PROGRAM MAIN
VAR
	work_number	: ULINT;
	act_dc_time : T_DCTIME64;
	dc_task_time : T_DCTIME64;
	dc_tick_time : T_DCTIME64;
	diff_time : T_DCTIME64;
	fbConvertDcTimeToPos : ConvertDcTimeToPos;
	position_at_task_start_point : LREAL;
	position_diff : LREAL;
	dc_time_array : ARRAY [0..1] OF T_DCTIME32;
	
	fb_timezone_info : FB_GetTimeZoneInformation := (bExecute := TRUE);
	event_messages : ARRAY [1..3] OF STRING;
	
	fbPower1:mc_power;
	fbPower2:mc_power;
	fbStop	: MC_Stop;
	fbGearOut : MC_GearOut;
	fbReset	: MC_Reset;
	
	stop_job : FB_Executor;
	basic_job : FB_Executor;
	demo_job : FB_Executor;
	gear_in_job : FB_Executor;
	gear_out_job : FB_Executor;
	init_pos_job : FB_Executor;
	jog_plus_job : FB_Executor;
	jog_minus_job : FB_Executor;
	fb_observer : FB_Observer;
	job_reset : BOOL;
	
	mc_power_future_creator: FutureMCPowerCreator;
	mc_reset_future_creator: FutureMCResetCreator;
	mc_set_position_future_creator: FutureMCSetPositionCreator;
	mc_inching_future_creator : FutureMCInchingCreator;
	mc_gear_in_future_creator : FutureMCGearInCreator;
	mc_gear_out_future_creator : FutureMCGearOutCreator;
	mc_move_rel_future_creator : FutureMCMoveRelativeCreator;
	mc_move_abs_future_creator : FutureMCMoveAbsoluteCreator;
	mc_move_velocity_future_creator: FutureMCMoveVelocityCreator;
	mc_stop_future_creator: FutureMCStopCreator;
	sleep_creator : FutureSleepCreator;

	
	iState:UINT;
	stopState : UINT;
	stAxis1:axis_ref;
	stAxis2:axis_ref;
	bStart: BOOL;
	bJogPlus: BOOL;
	bJogMinus: BOOL;
	bPower: BOOL;
	_bPower :BOOL;
	bPowerOn : BOOL;
	iPowerState : UINT;
	bReset:BOOL;
	bError:BOOL;
	bAllAxisPowerOn: BOOL;
	bInsync:BOOL;
	create_container: INT;
	boot_up : BOOL := TRUE;
	i: UINT;
	
	quit: INT;	
END_VAR

// Update state data for axis_ref.Status structure.
stAxis1.ReadStatus();
stAxis2.ReadStatus();

act_dc_time := F_GetActualDcTime64();
dc_task_time := F_GetCurDcTaskTime64();
dc_tick_time := F_GetCurDcTickTime64();

MEMCPY(ADR(dc_time_array), ADR(dc_task_time), SIZEOF(dc_task_time));

fbConvertDcTimeToPos(nAxisId := 1, nSubIdx := 16#10000, dcTime := dc_time_array[0] + 300000);
position_at_task_start_point := fbConvertDcTimeToPos.fPosition;
position_diff := stAxis1.NcToPlc.ActPos - fbConvertDcTimeToPos.fPosition;

diff_time := act_dc_time - dc_task_time;

IF boot_up THEN
	(*
	Initial setting at the time of starting PLC.
	*)
	
	// Creating basic running job container instance
	basic_job.create_container(ContainerType.PARALLEL_QUEUE, 'BASIC');
	// Enable continuous mode : Continue running job after all queued jobs are purged.
	basic_job.continuous_mode := TRUE;
	// Set top level job name
	basic_job.id := 'M1';
	// Set observer object: for event logging, IoT
	basic_job.job_event_reporter := fb_observer;
	// Create position initialization job.
	JobCreate_PosInit(init_pos_job);
	// Create gear-in job.
	JobCreate_GearIn(gear_in_job);
	// Create demo job.
	JobCreateDemo(demo_job);
	// Create inching job
	mc_inching_future_creator.set_parameters(stAxis2, TRUE,1 , 100);
	jog_plus_job.create_future(mc_inching_future_creator,'JOG_PLUS');
	
	mc_inching_future_creator.set_parameters(stAxis2, FALSE, 1, 100);		
	jog_minus_job.create_future(mc_inching_future_creator,'JOG_MINUS');

	boot_up := FALSE;
END_IF

// Power control
// Power off after gear decoupled and job unlinked.

IF NOT bPower THEN
	CASE stopState OF
		0: // Forced stop if any jobs are working.
			IF bPowerOn THEN
				IF stAxis1.Status.HasJob THEN
					fbStop(Axis := stAxis1, Execute := TRUE);
				ELSE
					fbStop(Axis := stAxis1, Execute := FALSE);
					IF NOT fbStop.Busy THEN
						stopState := 1;
					END_IF
				END_IF
			END_IF
		1: // make job state abort
			IF basic_job.abort() THEN
				stopState := 2;	
			END_IF
		2: // Decouple stAxis2 from stAxis1.
			IF stAxis2.Status.Coupled THEN
				fbGearOut(Slave := stAxis2,Execute := TRUE);
			ELSE
				fbGearOut(Slave := stAxis2,Execute := FALSE);
				stopState := 3;
			END_IF
		3: // Unlink machie jobs and reset state machine. 
			IF basic_job.reset(FALSE) THEN
				IF basic_job.init() THEN
					bPowerOn := FALSE;
					bStart := FALSE;
					stopState := 0;
					iState := 0;
				END_IF
			END_IF	
	END_CASE
END_IF

IF bPower AND NOT _bPower THEN
	bPowerOn := TRUE;
END_IF

_bPower := bPower;

fbPower1(Axis := stAxis1, Enable := bPowerOn, Enable_Positive := TRUE, Enable_Negative := TRUE, Override := 100.0);
fbPower2(Axis := stAxis2, Enable := bPowerOn, Enable_Positive := TRUE, Enable_Negative := TRUE, Override := 100.0);

CASE iState OF
	0: // Position reset after Power ON
		IF fbPower1.Status AND fbPower2.Status THEN
			init_pos_job.init();
			basic_job.children.append_job(init_pos_job);
			iState := 1;
		END_IF
	1: // Vacant
		IF init_pos_job.done THEN
			iState := 2;
		END_IF
	2: // Adjustment coupling position between each gear, and to be start.
		IF bJogPlus THEN
			IF jog_plus_job.init() THEN
				basic_job.children.append_job(jog_plus_job);
				bJogPlus := FALSE;				
			END_IF
		END_IF
		
		IF bJogMinus THEN
			IF jog_minus_job.init() THEN
				basic_job.children.append_job(jog_minus_job);
				bJogMinus := FALSE;				
			END_IF
		END_IF

		IF bStart THEN
				IF NOT stAxis2.Status.Coupled THEN
					IF gear_in_job.init() THEN
						basic_job.children.append_job(gear_in_job);
						iState := 3;
					END_IF
				ELSE
					iState := 3;
				END_IF
		END_IF
	3: // Setting working job ID into demo_job instance and append it as machine job.
		IF demo_job.init() THEN
			work_number := work_number + 1;
			demo_job.id := TO_STRING(work_number);
			basic_job.children.append_job(demo_job);
			iState := 4;
		END_IF
	4: // Decision to finish or to rerun demo_job by Start button.
		IF demo_job.done THEN
			IF bStart THEN
				iState := 3;
			ELSE
				iState := 1;
			END_IF
		END_IF
END_CASE

basic_job.execute();

bError := basic_job.nErrorID <> 0;

IF bReset THEN
	IF basic_job.error_reset() THEN
		IF basic_job.resume() THEN
			bReset := FALSE;
		END_IF
	END_IF 
END_IF

fbReset(Axis := stAxis1, Execute := bReset);
fbReset(Axis := stAxis2, Execute := bReset);


IF basic_job.ready THEN
	basic_job.start();
END_IF

// Event string

IF fb_observer.job_event_report.new_state = TO_STRING(E_FutureExecutionState.process) THEN
	event_messages[1] := SYSTEMTIME_TO_STRING(FILETIME64_TO_SYSTEMTIME(fb_observer.job_event_report.record_time));
	event_messages[2] := fb_observer.job_event_report.future_name;
	event_messages[3] := fb_observer.job_event_report.job_id;
END_IF

METHOD Execution : BOOL
VAR_INPUT
	main_job : REFERENCE TO FB_Executor;
	bStart : BOOL := TRUE;
END_VAR
Execution := main_job.execute();

IF main_job.ready THEN
	main_job.start();
END_IF

IF bStart THEN
	main_job.start();
END_IF
END_METHOD

METHOD JobCreate_GearIn : BOOL
VAR_INPUT
	job : REFERENCE TO FB_Executor;
END_VAR
// Gear In
mc_gear_in_future_creator.set_parameters(stAxis1, stAxis2);
job.create_future(mc_gear_in_future_creator,'Gear IN');
END_METHOD

METHOD JobCreate_GearOut : BOOL
VAR_INPUT
	job : REFERENCE TO FB_Executor;
END_VAR
// Gear In
mc_gear_out_future_creator.set_parameters(stAxis2);
job.create_future(mc_gear_out_future_creator,'Gear OUT');
END_METHOD

METHOD JobCreate_PosInit : BOOL
VAR_INPUT
	job : REFERENCE TO FB_Executor;
END_VAR
VAR
	_job_temp	: REFERENCE TO FB_Executor; // reference to job object for working.
END_VAR
job.create_container(ContainerType.PARALLEL, 'INIT_POS');
// position set to 0
mc_set_position_future_creator.set_parameters(stAxis1, 0);
_job_temp REF= job.children.create_job(mc_set_position_future_creator,'AXIS1_POS_INIT');

mc_set_position_future_creator.set_parameters(stAxis2, 0);
_job_temp REF= job.children.create_job(mc_set_position_future_creator,'AXIS2_POS_INIT');
END_METHOD

METHOD JobCreate_Power : BOOL
VAR_INPUT
	power_on_job : REFERENCE TO FB_Executor;
	power_off_job : REFERENCE TO FB_Executor;
END_VAR
VAR
	_job_temp	: REFERENCE TO FB_Executor; // reference to job object for working.
END_VAR
power_on_job.create_container(ContainerType.PARALLEL, 'POWER_ON');
power_off_job.create_container(ContainerType.PARALLEL, 'POWER_OFF');
// position set to 0
mc_power_future_creator.set_parameters(stAxis1, TRUE);
power_on_job.children.create_job(mc_power_future_creator,'AXIS1_POWER_ON');
mc_power_future_creator.set_parameters(stAxis2, TRUE);
power_on_job.children.create_job(mc_power_future_creator,'AXIS2_POWER_ON');

mc_power_future_creator.set_parameters(stAxis1, FALSE);
power_off_job.children.create_job(mc_power_future_creator,'AXIS1_POWER_OFF');
mc_power_future_creator.set_parameters(stAxis2, FALSE);
power_off_job.children.create_job(mc_power_future_creator,'AXIS2_POWER_OFF');
END_METHOD

METHOD JobCreate_Stop : BOOL
VAR_INPUT
	job : REFERENCE TO FB_Executor;
END_VAR
mc_stop_future_creator.set_parameters(stAxis1,0,0);
job.create_future(mc_stop_future_creator,'STOP');
END_METHOD

METHOD JobCreateDemo : BOOL
VAR_INPUT
	base_job : REFERENCE TO FB_Executor;
END_VAR
VAR
	_job_temp : REFERENCE TO FB_Executor;
	_job_temp_parent : REFERENCE TO FB_Executor;
	sleep : POINTER TO FutureSleep;
	sleep_creator : FutureSleepCreator;

	mc_move_rel_future : POINTER TO FutureMCMoveRelative;
	mc_move_rel_future_creator : FutureMCMoveRelativeCreator;

	mc_move_abs_future : POINTER TO FutureMCMoveAbsolute;
	mc_move_abs_future_creator : FutureMCMoveAbsoluteCreator;

	mc_move_velocity_future: POINTER TO FutureMCMoveVelocity;
	mc_move_velocity_future_creator: FutureMCMoveVelocityCreator;

END_VAR
base_job.create_container(ContainerTYpe.BATCH, 'DEMO_JOB');
// Sequence
_job_temp_parent REF= base_job.children.create_container(ContainerTYpe.BATCH, 'STEP MOVING');
FOR i := 1 TO 10 DO

	mc_move_rel_future_creator.set_parameters(stAxis1,20,200,0,0,0,0);
	_job_temp REF= _job_temp_parent.children.create_job(mc_move_rel_future_creator,'Move +20 deg, 200 deg/s');

	sleep_creator.sleep_time := T#100MS;
	_job_temp REF= _job_temp_parent.children.create_job(sleep_creator,'Wait 100ms');
	
END_FOR

// position set to 0

mc_move_abs_future_creator.set_parameters(stAxis1,0,200,0,0,0,0);
_job_temp REF= base_job.children.create_job(mc_move_abs_future_creator,'Back to home');

FOR i := 1 TO 10 DO

	mc_move_rel_future_creator.set_parameters(stAxis1,-20,200,0,0,0,0);
	_job_temp REF= base_job.children.create_job(mc_move_rel_future_creator,'Move -20 deg, 200 deg/s');

	sleep_creator.sleep_time := T#100MS;
	_job_temp REF= base_job.children.create_job(sleep_creator,'Wait 100ms');
	
END_FOR

// position to 0

mc_move_abs_future_creator.set_parameters(stAxis1,0,200,0,0,0,0);
_job_temp REF= base_job.children.create_job(mc_move_abs_future_creator,'Back to home');

sleep_creator.sleep_time := T#100MS;
_job_temp REF= base_job.children.create_job(sleep_creator,'Wait 100ms');

// 1000deg/s -> 500deg/s

mc_move_velocity_future_creator.set_parameters(stAxis1,MC_Direction.MC_Positive_Direction,1000,0,0,0,0);
_job_temp REF= base_job.children.create_job(mc_move_velocity_future_creator,'Move velocity');

sleep_creator.sleep_time := T#5S;
_job_temp REF= base_job.children.create_job(sleep_creator,'1000 deg/s 5 seconds');

mc_move_velocity_future_creator.set_parameters(stAxis1,MC_Direction.MC_Positive_Direction,500,0,0,0,0);
_job_temp REF= base_job.children.create_job(mc_move_velocity_future_creator,'Move velocity');

sleep_creator.sleep_time := T#5S;
_job_temp REF= base_job.children.create_job(sleep_creator,'500 deg/s 5 seconds');

mc_move_velocity_future_creator.set_parameters(stAxis1,MC_Direction.MC_Positive_Direction,250,0,0,0,0);
_job_temp REF= base_job.children.create_job(mc_move_velocity_future_creator,'Move velocity');

sleep_creator.sleep_time := T#5S;
_job_temp REF= base_job.children.create_job(sleep_creator,'250 deg/s 5 seconds');


mc_stop_future_creator.set_parameters(stAxis1,0,0);
_job_temp REF= base_job.children.create_job(mc_stop_future_creator,'STOP');

// position to 0

mc_move_abs_future_creator.set_parameters(stAxis1,0,1000,0,0,0,0);
_job_temp REF= base_job.children.create_job(mc_move_abs_future_creator,'Back to home');
END_METHOD

END_PROGRAM

(* stored: Version 1.1.0.1, ProductVersion 3.1.4024.12
   POU MAIN: Id {22afa678-1e60-4864-9c5a-6f323d8f260f}, SpecialFunc None
   Method Execution: Id {d52dbacd-3d99-403b-bb01-e4478be4b44b}
   Method JobCreate_GearIn: Id {fcc86729-849d-4b88-bffd-35052ffdfb89}
   Method JobCreate_GearOut: Id {8481b2d7-af94-4ac5-a0a7-0d042155ce39}
   Method JobCreate_PosInit: Id {8ecc2f01-c3e3-4110-a58b-a3226565c5d4}
   Method JobCreate_Power: Id {18a6dd20-4504-4367-a000-7e9c44ad113a}
   Method JobCreate_Stop: Id {1ad0fcd6-0e50-425e-8238-352c792d91f9}
   Method JobCreateDemo: Id {c6c18e30-8bba-4c6d-806d-02b28dd2a277} *)
